{attribute addProperty BoxType "EP2809-0042-0017"}
{attribute addProperty Id "DO_X01_PinAT %Q*ARRAY[0..1] OF DO_X01_Pin_7F374EB0429496728842949672950DO_X02_PinAT %Q*ARRAY[0..1] OF DO_X02_Pin_7F374EB0429496728842949672950DO_X03_PinAT %Q*ARRAY[0..1] OF DO_X03_Pin_7F374EB0429496728842949672950DO_X04_PinAT %Q*ARRAY[0..1] OF DO_X04_Pin_7F374EB0429496728842949672950DO_X05_PinAT %Q*ARRAY[0..1] OF DO_X05_Pin_7F374EB0429496728842949672950DO_X06_PinAT %Q*ARRAY[0..1] OF DO_X06_Pin_7F374EB0429496728842949672950DO_X07_PinAT %Q*ARRAY[0..1] OF DO_X07_Pin_7F374EB0429496728842949672950DO_X08_PinAT %Q*ARRAY[0..1] OF DO_X08_Pin_7F374EB0429496728842949672950WcStateAT %I*WcState_64F6A8C6810InfoDataAT %I*InfoData_192954DE1620"}
{attribute addProperty CRC "2752820038"}
{attribute addProperty SizeInBites "4294967256"}
{attribute addProperty SizeInBytes "34359738363"}
TYPE EP2809_713014EC :
STRUCT
	{attribute addProperty Name "DO_X01_Pin"}
	DO_X01_Pin : ARRAY[0..1] OF DO_X01_Pin_7F374EB0;
	{attribute addProperty Name "DO_X02_Pin"}
	DO_X02_Pin : ARRAY[0..1] OF DO_X02_Pin_7F374EB0;
	{attribute addProperty Name "DO_X03_Pin"}
	DO_X03_Pin : ARRAY[0..1] OF DO_X03_Pin_7F374EB0;
	{attribute addProperty Name "DO_X04_Pin"}
	DO_X04_Pin : ARRAY[0..1] OF DO_X04_Pin_7F374EB0;
	{attribute addProperty Name "DO_X05_Pin"}
	DO_X05_Pin : ARRAY[0..1] OF DO_X05_Pin_7F374EB0;
	{attribute addProperty Name "DO_X06_Pin"}
	DO_X06_Pin : ARRAY[0..1] OF DO_X06_Pin_7F374EB0;
	{attribute addProperty Name "DO_X07_Pin"}
	DO_X07_Pin : ARRAY[0..1] OF DO_X07_Pin_7F374EB0;
	{attribute addProperty Name "DO_X08_Pin"}
	DO_X08_Pin : ARRAY[0..1] OF DO_X08_Pin_7F374EB0;
	{attribute addProperty Name "WcState"}
	WcState : WcState_64F6A8C6;
	{attribute addProperty Name "InfoData"}
	InfoData : InfoData_192954DE;
END_STRUCT
END_TYPE

(* stored: Version 1.2.0.0, ProductVersion 3.1.4024.9
   DUT EP2809_713014EC: Id {e0f6ae01-1fde-4cfd-b882-9ff6cc25ea8c} *)
